FUNCTION_BLOCK FB_DeviceDWord EXTENDS FB_LinkDataDWord
VAR_INPUT		
	nControl  			: BYTE;
	nControlData 		: DWORD;
END_VAR

VAR_OUTPUT
	nStatus  			: BYTE;
	nStatusData  		: DWORD;
END_VAR

SUPER^();
Control := nControl;
ControlData := nControlData;
nStatus := Status;
nStatusData := StatusData;

END_FUNCTION_BLOCK

(* stored: Version 1.1.0.1, ProductVersion 3.1.4024.12
   POU FB_DeviceDWord: Id {03098450-d7fc-064d-1fa2-276c7d34d134}, SpecialFunc None *)
